(* PLC project Tc2_Utilities.FB_EnumFindFileList Demo, tc3-libraries-kb TwinCAT 3.1 *)
(* stored: creationDateTime 2026-05-11T00:00:00, modificationDateTime 2026-05-11T00:00:00 *)

PROGRAM P_Demo_FB_EnumFindFileList
  VAR
    fbFB_EnumFindFileList : FB_EnumFindFileList;  (* FB_EnumFindFileList 实例 *)
    bExec : BOOL := FALSE;
    sPattern : STRING := 'C:\\TwinCAT\\Boot\\*.config';
    aFiles : ARRAY[0..63] OF ST_FindFileEntry;
    nCount : UDINT;
    bBusy_ : BOOL;
    bErrFlag : BOOL;
    nErrCode : UDINT;
  END_VAR

// =============================================================================
// 场景：批量列文件。
// 价值：一次完成。
// 验证：触发后 aFiles 数组填入文件名，nCount 给数量。
// 验证步骤：
//   1. 右键 PLC 项目 → Import PLCopenXML → 选本文件
//   2. 引用 Tc2_Utilities（References → Add library）
//   3. 编译 → 登录 → 运行；按上方『验证』行的指示在线写值观察
// =============================================================================

fbFB_EnumFindFileList(
    bExecute := bExec, sPathName := sPattern, ePath := PATH_GENERIC,
    pAddr := ADR(aFiles), cbAddr := SIZEOF(aFiles), tTimeout := DEFAULT_ADS_TIMEOUT,
    nFileCnt => nCount, bBusy => bBusy_, bError => bErrFlag, nErrId => nErrCode
);
END_PROGRAM
